Universal Robots PolyScope program: rotate_90.urp

Program rotate_90 (installation=default directory=/programs/usbdisk/programs createdIn=5.12.4.1101661 lastSavedIn=5.12.4.1101661 robotSerialNumber=20225502378)
Calibrated DH parameters: a=[0.00022, -0.425328, -0.389701, 0.000059, 0.000065, 0]; d=[0.162608, 0.803456, 9.992211, -10.662202, 0.099702, 0.099559]; alpha=[1.570756, 0.001543, 0.004316, 1.570651, -1.570122, 0]; deltaTheta=[0, 0.002917, 0.116094, -0.119008, 0, -0.000001]
Robot Program (runOnlyOnce=true)
  tile_pos_id := 11
  num_rotations := 1
  rotated := 0
  ter_hover_pos := p[0,0,0,0,0,0]
  ter_lower_pos := p[0,0,0,0,0,0]
  ter_hov_rotated := p[0,0,0,0,0,0]
  ter_hov_move := p[0,0,0,0,0,0]
  ter_low_rotated := p[0,0,0,0,0,0]
  Script file /programs/DND/rot_ter_offset.script
    | ter_tile_row = (floor(tile_pos_id / 10)) - 1
    | ter_tile_col = (tile_pos_id % 10) - 1
    | 
    | ter_hover_offset = p[-0.088*ter_tile_row, -0.088*ter_tile_col,0,0,0,0]
    | 
    | ter_hover_pos = pose_add(ter_base_hover, ter_hover_offset)
    | ter_lower_pos = pose_add(ter_hover_pos, p[0,0,-0.109,0,0,0])
    | 
    | ter_hov_rotated= pose_trans(ter_hover_pos, p[0,0,0,0,0,1.5708])
    | ter_hov_move= pose_add(ter_hov_rotated, p[-0.021, -0.0656, 0, 0, 0, 0])
    | ter_low_rotated = pose_add(ter_hov_move, p[0,0,-0.102,0,0,0])
  Loop While (checkContinuously=true) expression=rotated < num_rotations
    MoveL speed 250 mm/s, acceleration 1200 mm/s^2 (useActiveTCP=true) feature=Base
      Waypoint Waypoint (Variable): variable=ter_hover_pos
    URCap Gripper (Robotiq_Grippers, Robotiq Inc.) dataModel(position=75.0, force=0.0, speed=0.0, positionInDouble=75.0, forceInDouble=0.0, speedInDouble=0.0, slaveIds=[9], blocking=true)
    MoveL speed 250 mm/s, acceleration 1200 mm/s^2 (useActiveTCP=true) feature=Base
      Waypoint Waypoint (Variable): variable=ter_lower_pos
    URCap Gripper (Robotiq_Grippers, Robotiq Inc.) dataModel(position=100.0, force=0.0, speed=0.0, positionInDouble=100.0, forceInDouble=0.0, speedInDouble=0.0, slaveIds=[9], blocking=true)
    MoveL speed 250 mm/s, acceleration 1200 mm/s^2 (useActiveTCP=true) feature=Base
      Waypoint Waypoint (Variable): variable=ter_hover_pos
      Waypoint Waypoint (Variable): variable=ter_hov_rotated
      Waypoint Waypoint (Variable): variable=ter_hov_move
      Waypoint Waypoint (Variable): variable=ter_low_rotated
    URCap Gripper (Robotiq_Grippers, Robotiq Inc.) dataModel(position=75.0, force=0.0, speed=0.0, positionInDouble=75.0, forceInDouble=0.0, speedInDouble=0.0, slaveIds=[9], blocking=true)
    MoveL speed 250 mm/s, acceleration 1200 mm/s^2 (useActiveTCP=true) feature=Base
      Waypoint Waypoint (Variable): variable=ter_hov_move
    rotated := rotated + 1
